Staubli VAL3: onExit.pgx

program onExit(bool x_bSave)
  local string l_sMessage
  local bool l_bYes
  local num l_nResult
begin
  if x_bSave
    // ask to save
    //    call language:message(l_sMessage,-1)
    //    call use:yes_no(l_sMessage,l_bYes)
    //    if l_bYes
    call tcp:save(l_nResult)
    // send back the gun
    //    endIf
  endIf
  // give back and update
  saveData:nIndexTool=nIndexTool
  call tcp:getTool(saveData:tTool,nIndexTool)
end
